Fanuc KAREL source: kf00047.KL

-- PROVISIONAL review KL for V940-1; original PC SHA256 51e3c29baddb6bcefebefb01b134ae82c560810600f1294c94d89b753f8cff6c
-- Incomplete behavior may be omitted. Consult companion uncertainty JSON. Do not deploy.
PROGRAM KF00047
%NOLOCKGROUP
VAR
  I : INTEGER
  J : INTEGER
  X : REAL
  Y : REAL
  B : BOOLEAN
  C : BOOLEAN
  TXT : STRING[80]
  TXT2 : STRING[80]
  STATUS : INTEGER
-- UNRESOLVED_DECL AI type=002010
-- UNRESOLVED_DECL BI type=002010
-- UNRESOLVED_DECL P type=000102
-- UNRESOLVED_DECL JP type=000199
-- UNRESOLVED_DECL PF type=000101
-- UNRESOLVED_DECL V1 type=000013
-- UNRESOLVED_DECL V2 type=000013
BEGIN
  -- V9_EQ_BRANCH_SUBREGION_HINT bounded four-record physical order; branch ownership/target, source/runtime/producer release held
  -- V9_EXPOSED_INDEXED_TABLE_HINT layout=0001; 2 counted words exposed once; source arms/runtime held
  -- UNRESOLVED_PC offsets 5-12; opcodes 9D,23
  -- UNRESOLVED_PC offsets 17-28; opcodes 2E,23
  -- UNRESOLVED_PC offsets 33-46; opcodes 21,9D,57,79
  -- UNRESOLVED_PC offsets 51-68; opcodes 21,2E,57,79
  -- UNRESOLVED_PC offsets 73-84; opcodes 2E,23
  -- UNRESOLVED_PC offsets 99-103; opcodes 7F
END KF00047
